(* PLC project modemanagement, Dassault Systèmes ControlBuild 2024x Refresh1 *)
(* stored: creationDateTime 2024-04-16T09:45:42-01:00 *)

FUNCTION_BLOCK flask_motion_app.modemanagement
  VAR_INPUT
    bpStart : BOOL := false;
    bpAuto : BOOL := false;
    bpManu : BOOL := false;
    bpEmergencyStop : BOOL := false;
    bpStop : BOOL := false;
  END_VAR
  VAR_OUTPUT
    Auto : BOOL := false;
    Manu : BOOL := false;
    run : BOOL := false;
  END_VAR

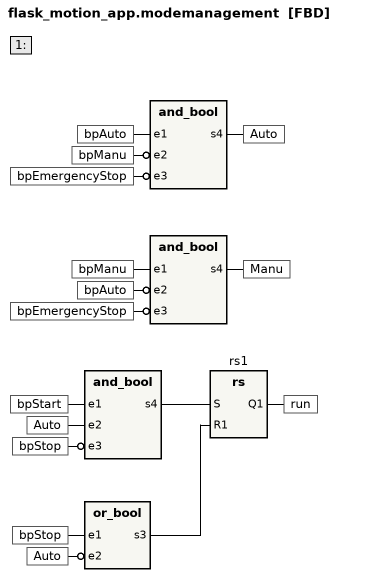
(* FBD diagram, written out as Structured Text *)
1:
Auto := and_bool(bpAuto, NOT bpManu, NOT bpEmergencyStop);
Manu := and_bool(bpManu, NOT bpAuto, NOT bpEmergencyStop);
rs1(S := and_bool(bpStart, Auto, NOT bpStop), R1 := or_bool(bpStop, NOT Auto));
run := rs1.Q1;
END_FUNCTION_BLOCK
